FUNCTION_BLOCK CU020ExampleCompositComponent EXTENDS TcoCore.TcoComponent
VAR_INPUT
END_VAR
VAR_OUTPUT
END_VAR
VAR
END_VAR

END_FUNCTION_BLOCK

(* stored: Version 1.1.0.1
   POU CU020ExampleCompositComponent: Id {e7415cd4-fbeb-4cf7-9b65-d3436cf3b7b9}, SpecialFunc None *)
